TYPE ST_GroupBaseEmulation :
(**************************************************************************************
 * 	Application		:	BoxControl Framework
 *	Revision		:	$Revision: 404529 $
 *	Revision date	:	$Date: 2018-04-23 08:21:38 +0200 (Mo., 23 Apr 2018) $
 *	Last changed by	:	$Author: b7bolm $
 *	URL				:	$URL: http://almscdc.swisslog.com/repo/SWPD/Development/BoxControlFramework/20_Release/trunk/01_Software/BCF/BCF/JumpStart/20_Product/11_Emu/14_Groups/10_Lib/10_Conv/01_DUTs/ST_GroupBaseEmulation.TcDUT $
 *
 *	Purpose			:	Function interface - Contains data which is provided by the
 *						function or is input from other objects.
 *
 * ------------------------------------------------------------------------------------
 *	Copyright Swisslog [IP AG], Switzerland. All rights reserved.
 * 
 * ------------------------------------------------------------------------------------
 *	
 * 	Revision History: 
 *
 * 	VERSION			DATE			INITIALS			DESCRIPTION
 *	0.1				01.01.2001		swl					Example
 *
 **************************************************************************************)
STRUCT
	rGroupDataReal				: REFERENCE TO ST_GroupData;
	GroupDataEmpty				: ST_GroupData;
	rGroupInterfaceReal			: REFERENCE TO ST_GroupInterface;
	GroupInterfaceEmpty			: ST_GroupInterface;
	rSettingsGroupReal			: REFERENCE TO ST_CFG_Group; 	
	SettingsGroupEmpty			: ST_CFG_Group;
	eMsgType					: E_ITC_MsgTypeConv;
	ERQ							: ST_ITC_ERQ;
END_STRUCT
END_TYPE

(* stored: Version 1.1.0.1, ProductVersion 3.1.4022.12
   DUT ST_GroupBaseEmulation: Id {e1d44f4a-7a54-468b-9ac2-a0b9bdc56e29} *)
